PROGRAM MAIN
VAR
	App : App;
END_VAR

App.Run();

END_PROGRAM

(* stored: Version 1.1.0.1, ProductVersion 3.1.4024.9
   POU MAIN: Id {a6a9e387-99f0-45b6-a90d-d39641abce81}, SpecialFunc None *)
